Yaskawa INFORM job: AAA1.JBI

/JOB
//NAME AAA
//POS
///NPOS 103,0,0,0,0,0
///TOOL 10
///POSTYPE PULSE
///PULSE
C00000=-50133,3180,-14203,-13218,-96470,56018
C00001=-44932,-4570,-20740,-13991,-96319,55770
C00002=-44373,-5320,-21356,-14077,-96307,55735
C00003=-43832,-6151,-22025,-14192,-96254,55715
C00004=-43312,-7063,-22747,-14335,-96161,55710
C00005=-42811,-8059,-23522,-14506,-96028,55720
C00006=-42329,-9139,-24349,-14703,-95854,55745
C00007=-41867,-10304,-25229,-14925,-95640,55784
C00008=-41423,-11555,-26162,-15173,-95385,55837
C00009=-40997,-12894,-27148,-15445,-95091,55905
C00010=-40590,-14321,-28188,-15741,-94757,55986
C00011=-40201,-15836,-29281,-16060,-94385,56081
C00012=-39828,-17441,-30428,-16403,-93974,56189
C00013=-39473,-19134,-31627,-16768,-93526,56309
C00014=-39135,-20916,-32880,-17155,-93041,56442
C00015=-38812,-22786,-34185,-17564,-92522,56585
C00016=-38504,-24741,-35540,-17995,-91970,56739
C00017=-38211,-26781,-36945,-18445,-91386,56902
C00018=-37931,-28901,-38397,-18916,-90773,57072
C00019=-37662,-31098,-39893,-19405,-90134,57248
C00020=-37404,-33368,-41430,-19911,-89471,57428
C00021=-37154,-35704,-43005,-20434,-88788,57608
C00022=-36910,-38100,-44612,-20972,-88087,57787
C00023=-36670,-40550,-46247,-21523,-87373,57961
C00024=-36430,-43045,-47904,-22085,-86648,58127
C00025=-36189,-45575,-49576,-22656,-85917,58280
C00026=-35943,-48132,-51257,-23232,-85183,58417
C00027=-35688,-50704,-52939,-23812,-84450,58531
C00028=-35421,-53282,-54615,-24392,-83720,58620
C00029=-35138,-55853,-56276,-24970,-82996,58675
C00030=-34834,-58405,-57915,-25540,-82282,58693
C00031=-34506,-60927,-59522,-26100,-81580,58667
C00032=-34149,-63405,-61089,-26646,-80890,58591
C00033=-33758,-65825,-62606,-27173,-80215,58458
C00034=-33330,-68174,-64065,-27676,-79556,58263
C00035=-32858,-70436,-65455,-28149,-78914,57999
C00036=-32338,-72594,-66765,-28588,-78290,57660
C00037=-31764,-74630,-67985,-28985,-77683,57242
C00038=-31130,-76524,-69102,-29332,-77097,56740
C00039=-30432,-78253,-70102,-29621,-76531,56149
C00040=-29663,-79790,-70969,-29842,-75990,55469
C00041=-28817,-81107,-71687,-29985,-75478,54697
C00042=-27890,-82171,-72238,-30040,-75001,53836
C00043=-26877,-82945,-72600,-29996,-74567,52886
C00044=-25777,-83390,-72753,-29845,-74188,51855
C00045=-24589,-83463,-72673,-29579,-73880,50748
C00046=-23318,-83121,-72339,-29195,-73662,49577
C00047=-21970,-82322,-71729,-28696,-73554,48353
C00048=-20555,-81028,-70824,-28088,-73580,47088
C00049=-19089,-79208,-69608,-27384,-73767,45797
C00050=-17589,-76837,-68071,-26604,-74138,44495
C00051=-16073,-73906,-66211,-25772,-74716,43196
C00052=-14564,-70418,-64033,-24916,-75520,41915
C00053=-13081,-66394,-61552,-24067,-76559,40664
C00054=-11645,-61874,-58794,-23256,-77838,39457
C00055=-10271,-56916,-55801,-22510,-79345,38302
C00056=-8973,-51602,-52623,-21856,-81062,37211
C00057=-7761,-46025,-49324,-21312,-82954,36192
C00058=-6639,-40297,-45974,-20891,-84982,35254
C00059=-5608,-34529,-42644,-20599,-87095,34408
C00060=-4665,-28836,-39404,-20439,-89244,33667
C00061=-3804,-23314,-36313,-20407,-91383,33044
C00062=-3018,-18045,-33417,-20496,-93472,32556
C00063=-2299,-13094,-30751,-20698,-95480,32222
C00064=-1638,-8506,-28333,-21004,-97384,32063
C00065=-1026,-4306,-26170,-21403,-99174,32100
C00066=-453,-510,-24261,-21881,-100844,32352
C00067=93,2872,-22600,-22421,-102394,32835
C00068=626,5829,-21179,-23000,-103819,33558
C00069=1159,8338,-19993,-23587,-105111,34516
C00070=1709,10361,-19045,-24145,-106245,35686
C00071=2286,11842,-18345,-24634,-107183,37026
C00072=2903,12711,-17913,-25017,-107873,38476
C00073=3560,12885,-17781,-25267,-108251,39966
C00074=4257,12287,-17987,-25373,-108255,41425
C00075=4988,10851,-18576,-25338,-107832,42797
C00076=5751,8528,-19592,-25174,-106945,44045
C00077=6547,5286,-21081,-24900,-105572,45150
C00078=7382,1120,-23079,-24536,-103710,46106
C00079=8270,-3948,-25612,-24099,-101377,46915
C00080=9225,-9852,-28675,-23607,-98614,47582
C00081=10264,-16475,-32233,-23073,-95486,48105
C00082=11401,-23643,-36206,-22508,-92082,48476
C00083=12641,-31141,-40478,-21920,-88506,48676
C00084=13982,-38738,-44910,-21319,-84863,48674
C00085=15409,-46214,-49363,-20713,-81245,48432
C00086=16899,-53388,-53715,-20114,-77719,47903
C00087=18426,-60129,-57870,-19532,-74318,47034
C00088=19969,-66346,-61761,-18968,-71053,45765
C00089=21519,-71965,-65326,-18401,-67918,44036
C00090=23085,-76882,-68488,-17770,-64921,41795
C00091=24683,-80911,-71116,-16983,-62117,39041
C00092=26307,-83750,-73012,-15956,-59646,35864
C00093=27885,-85043,-73941,-14719,-57722,32479
C00094=29265,-84510,-73713,-13471,-56570,29191
C00095=30275,-82064,-72254,-12522,-56336,26293
C00096=30804,-77811,-69609,-12125,-57056,23962
C00097=30829,-71964,-65899,-12378,-58687,22231
C00098=30409,-64777,-61294,-13224,-61140,21030
C00099=29656,-56531,-55994,-14515,-64293,20234
C00100=28704,-47549,-50242,-16082,-67980,19722
C00101=27684,-38195,-44311,-17787,-72001,19406
C00102=21881,40354,769,-35317,-108423,13094
//INST
///DATE 2023/03/27 12:31
///ATTR SC,RW
///GROUP1 RB1
NOP
MOVJ C00000 VJ=5.0
MOVL C00001 V=400.0
MOVL C00002 V=400.0
MOVL C00003 V=400.0
MOVL C00004 V=400.0
MOVL C00005 V=400.0
MOVL C00006 V=400.0
MOVL C00007 V=400.0
MOVL C00008 V=400.0
MOVL C00009 V=400.0
MOVL C00010 V=400.0
MOVL C00011 V=400.0
MOVL C00012 V=400.0
MOVL C00013 V=400.0
MOVL C00014 V=400.0
MOVL C00015 V=400.0
MOVL C00016 V=400.0
MOVL C00017 V=400.0
MOVL C00018 V=400.0
MOVL C00019 V=400.0
MOVL C00020 V=400.0
MOVL C00021 V=400.0
MOVL C00022 V=400.0
MOVL C00023 V=400.0
MOVL C00024 V=400.0
MOVL C00025 V=400.0
MOVL C00026 V=400.0
MOVL C00027 V=400.0
MOVL C00028 V=400.0
MOVL C00029 V=400.0
MOVL C00030 V=400.0
MOVL C00031 V=400.0
MOVL C00032 V=400.0
MOVL C00033 V=400.0
MOVL C00034 V=400.0
MOVL C00035 V=400.0
MOVL C00036 V=400.0
MOVL C00037 V=400.0
MOVL C00038 V=400.0
MOVL C00039 V=400.0
MOVL C00040 V=400.0
MOVL C00041 V=400.0
MOVL C00042 V=400.0
MOVL C00043 V=400.0
MOVL C00044 V=400.0
MOVL C00045 V=400.0
MOVL C00046 V=400.0
MOVL C00047 V=400.0
MOVL C00048 V=400.0
MOVL C00049 V=400.0
MOVL C00050 V=400.0
MOVL C00051 V=400.0
MOVL C00052 V=400.0
MOVL C00053 V=400.0
MOVL C00054 V=400.0
MOVL C00055 V=400.0
MOVL C00056 V=400.0
MOVL C00057 V=400.0
MOVL C00058 V=400.0
MOVL C00059 V=400.0
MOVL C00060 V=400.0
MOVL C00061 V=400.0
MOVL C00062 V=400.0
MOVL C00063 V=400.0
MOVL C00064 V=400.0
MOVL C00065 V=400.0
MOVL C00066 V=400.0
MOVL C00067 V=400.0
MOVL C00068 V=400.0
MOVL C00069 V=400.0
MOVL C00070 V=400.0
MOVL C00071 V=400.0
MOVL C00072 V=400.0
MOVL C00073 V=400.0
MOVL C00074 V=400.0
MOVL C00075 V=400.0
MOVL C00076 V=400.0
MOVL C00077 V=400.0
MOVL C00078 V=400.0
MOVL C00079 V=400.0
MOVL C00080 V=400.0
MOVL C00081 V=400.0
MOVL C00082 V=400.0
MOVL C00083 V=400.0
MOVL C00084 V=400.0
MOVL C00085 V=400.0
MOVL C00086 V=400.0
MOVL C00087 V=400.0
MOVL C00088 V=400.0
MOVL C00089 V=400.0
MOVL C00090 V=400.0
MOVL C00091 V=400.0
MOVL C00092 V=400.0
MOVL C00093 V=400.0
MOVL C00094 V=400.0
MOVL C00095 V=400.0
MOVL C00096 V=400.0
MOVL C00097 V=400.0
MOVL C00098 V=400.0
MOVL C00099 V=400.0
MOVL C00100 V=400.0
MOVL C00101 V=400.0
MOVL C00102 V=400.0
END
